Staubli VAL3: cycle_doEvent.pgx

program cycle_doEvent(InstrItem x_iInstr (dimensions=1), num x_nIndex (dimensions=1))
  local ActionItem l_aAction
  local bool l_bTraj
  local num l_nId
  local num l_nOffset
  local num l_nResult
  local string l_sInstruction
  local string l_sName
  local string l_sPath
begin
  //
  // DIVIDE INTO trajectory or NOT
  //
  call saveData:getPathInstr(x_iInstr.sType,l_sPath)
  if l_sPath!=""
    // DIVIDE INSTRUCTION FROM TRAJECTORY
    if find(l_sPath,"trajectory")==-1
      // EXECUTE THE ACTION
      call action_wait()
      // UPDATE THE ACTION TO DO...
      l_aAction.nDistance=1-saveData:nRound/100
      call cycleStatus:getLastId(l_aAction.nMoveId)
      l_aAction.iInstr=x_iInstr
      l_aAction.nPointId=-1
      call action_do(l_aAction,x_nIndex)
    else
      // TRAJ
      // print the action log
      l_sInstruction=x_iInstr.sType+" "+x_iInstr.sData
      if cycleStatus:bCycle
        // set the clock end
        call cycleStatus:printLog("-"+l_sInstruction)
      endIf
      // update the LINE ID
      cycleStatus:nLastIdPoint=x_nIndex
      // run it
      call memory_onRun(x_iInstr)
    endIf
  else
    // PATH NOT FOUND
    cycleStatus:bToStop=true
  endIf
end
